# EPICS autosave request: iocBoot/generic_motors_ioc/dbSave/CCD_Lp_.req
%
% BURT Request File
%
% $(P)CCD:Lp:  CCD lateral position
%

file assy.req ASSY=$(P)CCD:Lp
$(P)CCD:Lp:Dmhmv
$(P)CCD:Lp:aH
$(P)CCD:Lp:mLink
file mtr1.req MTR1=$(P)CCD:ml
file drv1.req DRV1=$(P)CCD:DL
